Yaskawa INFORM job: u_test1TRJ0.JBI

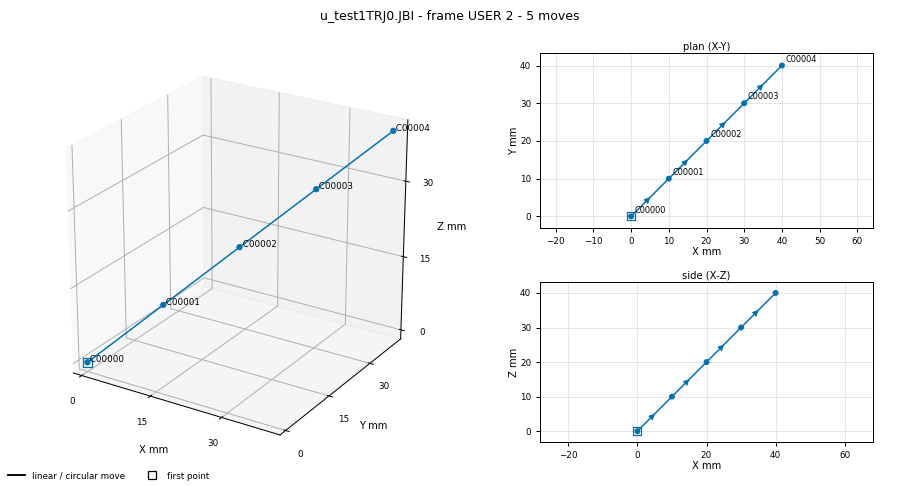
[picture p0: tool path of u_test1TRJ0.JBI in frame USER 2, 5 of 5 moves have a stored position in this frame; points joined in program order, loops and branches not executed]
/JOB
//NAME u_test1TRJ0
///FOLDERNAME DEMO
//POS
///NPOS 5,0,0,0,0,0
///USER 2
///TOOL 7
///POSTYPE USER
///RECTAN
///RCONF 1,0,0,0,0,0,0,0,0,0,0,0,0,0,0,0,0,0,0,0,0,0,0,0
C00000=0.000,0.000,0.000,-180.0000,0.0000,0.0000
C00001=10.000,10.000,10.000,-180.0000,0.0000,0.0000
C00002=20.000,20.000,20.000,-180.0000,0.0000,0.0000
C00003=30.000,30.000,30.000,-180.0000,0.0000,0.0000
C00004=40.000,40.000,40.000,-180.0000,0.0000,0.0000
//INST
///DATE 2021/09/21 16:22
///COMM
///ATTR SC,RW,RJ
////FRAME USER 2
///GROUP1 RB1
NOP
' first example of file for tool generation
SPEED V=10.2
MOVL C00000
SPEED V=50.0
MOVL C00001
MOVL C00002
TIMER T=10.23
DOUT OG#(12) 1
ARCON
MOVL C00003
ARCOF
MOVL C00004
END
